FUNCTION_BLOCK Director
VAR_INPUT
END_VAR
VAR_OUTPUT
END_VAR
VAR
END_VAR

END_FUNCTION_BLOCK

(* stored: Version 1.1.0.1, ProductVersion 3.1.4024.11
   POU Director: Id {7ba3b411-03e2-4744-bc96-6b241362c795}, SpecialFunc None *)
